INTERFACE ITF_GroupE_TE2_HMI EXTENDS ITF_BaseGroupElement_HMI

METHOD LinkGroupEData : BOOL
VAR_INPUT
	stData				: REFERENCE TO ST_GroupE_TE2_HMI_Link;
END_VAR
END_METHOD

END_INTERFACE

(* stored: Version 1.1.0.1, ProductVersion 3.1.4024.15
   Itf ITF_GroupE_TE2_HMI: Id {3050dc31-db2c-4ea8-abc2-4dae72fd190a}
   Method LinkGroupEData: Id {e3bf014b-9cc1-47a2-b50a-0ad79fcb2c79} *)
